PROGRAM MAIN
VAR
	BottleTester : fb_BottleTester_Main;
END_VAR

BottleTester ();

END_PROGRAM

(* stored: Version 1.1.0.1
   POU MAIN: Id {bbc2608b-f0e9-4100-9c8d-3931d6a0ecb9}, SpecialFunc None *)
